KUKA KRL program: start_weld_geo.src

&ACCESS RVO3
&REL 149
&COMMENT start_weld_GEO
&PARAM DISKPATH = KRC:\R1\Program\SubRotinas
DEF start_weld_GEO( )
;
; INICIO DE SOLDA COM GOEOMETRIA
;FOLD OUT 3338 'R4 solda geometria concluida' State=FALSE ;%{PE}%R 8.2.20,%MKUKATPBASIS,%COUT,%VOUTX,%P 2:3338, 3:R4 solda geometria concluida, 5:FALSE, 6:
$OUT[3338]=FALSE
;ENDFOLD
;
END
